# EPICS StreamDevice protocol: riesling/riesling_spaetlese/device_config/riesling_spaetlese.proto
Terminator = LF;
ExtraInput = Ignore;

#Optionale Zusatzbefehle:
#version{out "v"; in "%39c";}
#range_auto{ out "a"; in "range auto";}
#range_fine{ out "0"; in "range 0";}
#range_coarse{ out "1"; in "range 1";}

read {
	in "r %d";
}
